{attribute 'pack_mode' := '1'}
TYPE MoveAxisRelative EXTENDS IncomingMessage :
STRUCT
	axisIndex: DINT; (* 1 or 2.*)
	distance: LREAL;
	moveTime: TIME;
END_STRUCT
END_TYPE

(* stored: Version 1.1.0.1, ProductVersion 3.1.4022.12
   DUT MoveAxisRelative: Id {05d30087-dc30-4e15-9f19-3c8d74281187} *)
